FUNCTION Convert_LINT_TO_LREAL : Hresult
VAR_INPUT
	in : LINT;
	out : REFERENCE TO LREAL;
END_VAR
VAR
	converted : LREAL;
END_VAR

converted := LINT_TO_LREAL(in);

IF (LREAL_TO_LINT(converted) <> in) THEN
	Convert_LINT_TO_LREAL := INCOMPATIBLE;
	RETURN;
END_IF

out := converted;

END_FUNCTION

(* stored: Version 1.1.0.1, ProductVersion 3.1.4024.12
   POU Convert_LINT_TO_LREAL: Id {286ed6d9-0f52-499f-8d84-b050940e0c5f}, SpecialFunc None *)
